FUNCTION_BLOCK FB_Rechazar_SFC

VAR_INPUT
    // SFC-Flags
    SFCPause: BOOL;
    SFCReset: BOOL;
    
    // Parametros de control de la estacion
    CicloACiclo: BOOL;    

	
	// Sincronizacion
    Benido: BOOL := TRUE;
    Ejecuta: BOOL;
	
    RechazadorDetras AT %I* : BOOL;
    RechazadorDelante AT %I* : BOOL;
    RechazadorArriba AT %I* : BOOL;
    RechazadorVacio AT %I* : BOOL;
END_VAR
VAR_OUTPUT
	
    Acabhe: BOOL;
    ListoKalisto: BOOL;

  //  RechazadorAvanza AT %Q* : BOOL;
  //  RechazadorRetrocede AT %Q* : BOOL;
    //RechazadorBaja AT %Q* : BOOL;
   // RechazadorSucciona AT %Q* : BOOL;
    
    RechazadorAvanza: BOOL;
    RechazadorRetrocede: BOOL;
    RechazadorBaja: BOOL;
    RechazadorSucciona: BOOL;
END_VAR
VAR
END_VAR

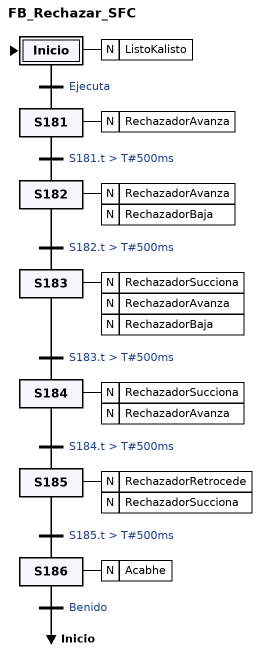
INITIAL_STEP Inicio:
    ListoKalisto(N);
END_STEP
TRANSITION FROM Inicio TO S181
    := Ejecuta;
END_TRANSITION
STEP S181:
    RechazadorAvanza(N);
END_STEP
TRANSITION FROM S181 TO S182
    := S181.t > T#500ms;
END_TRANSITION
STEP S182:
    RechazadorAvanza(N);
    RechazadorBaja(N);
END_STEP
TRANSITION FROM S182 TO S183
    := S182.t > T#500ms;
END_TRANSITION
STEP S183:
    RechazadorSucciona(N);
    RechazadorAvanza(N);
    RechazadorBaja(N);
END_STEP
TRANSITION FROM S183 TO S184
    := S183.t > T#500ms;
END_TRANSITION
STEP S184:
    RechazadorSucciona(N);
    RechazadorAvanza(N);
END_STEP
TRANSITION FROM S184 TO S185
    := S184.t > T#500ms;
END_TRANSITION
STEP S185:
    RechazadorRetrocede(N);
    RechazadorSucciona(N);
END_STEP
TRANSITION FROM S185 TO S186
    := S185.t > T#500ms;
END_TRANSITION
STEP S186:
    Acabhe(N);
END_STEP
TRANSITION FROM S186 TO Inicio
    := Benido;
END_TRANSITION

END_FUNCTION_BLOCK

(* stored: Version 1.1.0.1, ProductVersion 3.1.4024.12
   POU FB_Rechazar_SFC: Id {ac648ee0-fefe-40b1-ac92-2a6c7dc491a4}, SpecialFunc None *)
